# EPICS autosave request: motorSimApp/Db/sensor.req
$(P):sensor$(N).INPA
$(P):sensor$(N).INPB
